FUNCTION_BLOCK FB_Basis
VAR_INPUT
	// Betriebsvariablen
	eSysCommand				:eSystemCommand;
END_VAR
VAR_OUTPUT
END_VAR
VAR
	// Managementvariablen
	iState					:INT;
	
	// Transitionsvariablen
	bStart					:BOOL;
	bBeendet 				:BOOL;
	bReset					:BOOL;
	
	// SFC-Flags
	SFCReset				:BOOL;
	SFCCurrentStep			:BOOL;
END_VAR

METHOD M_Reset : BOOL
VAR_INPUT
END_VAR
bReset := TRUE;
END_METHOD

METHOD M_Start : BOOL
VAR_INPUT
END_VAR
bBeendet := FALSE;
bStart := TRUE;
END_METHOD

METHOD M_Stop : BOOL
VAR_INPUT
END_VAR
bStart := FALSE;
bBeendet := TRUE;
END_METHOD

PROPERTY P_Finished : BOOL
GET
P_Finished := bBeendet;
END_GET
END_PROPERTY

PROPERTY P_State : INT;
GET
P_State := iState;
END_GET
END_PROPERTY

END_FUNCTION_BLOCK

(* stored: Version 1.1.0.1
   POU FB_Basis: Id {f85c9ba4-7c23-49dd-97a7-335305937fa5}, SpecialFunc None
   Folder 01_Steuerungsmethoden: Id {c078cb8f-4ec6-40ed-9e3e-dc504220165d}
   Folder 02_Steuerungseigenschaften: Id {dd619586-3472-4567-846d-1e7ffd186aea}
   Method M_Reset: Id {f2c3cb40-97ad-4b16-b682-86e7a7aa9936}
   Method M_Start: Id {3b8d54a5-f826-4c91-bb15-3ca6280995f7}
   Method M_Stop: Id {aeab132f-14e3-468c-af3a-a7afa26bb694}
   Property P_Finished: Id {a66d494a-965d-4cb7-82b2-665c252cc716}
   Get Get: Id {a1a0563e-e419-4637-b3d5-a4a7a86c2f9d}
   Property P_State: Id {424b331b-368b-4080-a1ab-e6d22be996db}
   Get Get: Id {7d3a29b1-e786-46aa-a0eb-253fc5114027} *)
